{attribute 'GeneratedUsingTerminal: EJ1101-0022-0016'}
{attribute addProperty BoxType "EJ1101-0022-0016"}
{attribute addProperty Id "EtcSlaveTerminalBaseWcStateAT %I*WcState_0B2B16F91InfoDataAT %I*InfoData_32EB74EA10"}
{attribute addProperty CRC "3076194958"}
{attribute addProperty Size "11"}
TYPE EJ1101_B75B028E EXTENDS EtcSlaveTerminalBase :
STRUCT
	{attribute addProperty Name "WcState"}
	WcState : WcState_0B2B16F9;
	{attribute addProperty Name "InfoData"}
	InfoData : InfoData_32EB74EA;
END_STRUCT
END_TYPE

(* stored: Version 1.2.0.0, ProductVersion 3.1.4024.9
   DUT EJ1101_B75B028E: Id {b4b5f600-b0f8-4208-a400-8fffbaee8d4d} *)
